TYPE ST_RejectReason_PK3_OUT3 :
STRUCT
	Reason	:STRING;
END_STRUCT
END_TYPE

(* stored: Version 1.1.0.1, ProductVersion 3.1.4024.13
   DUT ST_RejectReason_PK3_OUT3: Id {150db487-dab8-4a52-ad14-e5e1f24f7865} *)
